// TIA Portal project "scl_5" (V18)

(* hardware
DEVICE "S7-1200 station_1"  S7-1200 Station
   slot 0: "Rack_0"  S7-1200 Rack  Rack  V1.0
   slot 1: "PLC_1"  CPU 1214C DC/DC/DC  6ES7 214-1AG40-0XB0  V4.6
*)

// ===== PLC "PLC_1"  CPU 1214C DC/DC/DC =====

VAR_GLOBAL   // PLC tag table "Default tag table"
   "İLERİ START" AT %I0.0 : Bool;
   "GERİ START" AT %I0.1 : Bool;
   "STOP" AT %I0.2 : Bool;
   "MOTOR İLERİ" AT %Q0.0 : Bool;
   "MOTOR GERİ" AT %Q0.1 : Bool;
END_VAR

FUNCTION "Block_1" : Void   // FC1, SCL
{ S7_Optimized_Access := 'TRUE' }
VERSION : 0.1
BEGIN
   IF "İLERİ START" AND NOT "MOTOR GERİ"=1 THEN
       // Statement section IF

       "MOTOR İLERİ":=1;
   END_IF;
   IF "GERİ START" AND NOT "MOTOR İLERİ" = 1 THEN
       // Statement section IF

       "MOTOR GERİ" := 1;

   END_IF;
   IF "STOP"=1 THEN
       // Statement section IF

       "MOTOR İLERİ" := 0;
       "MOTOR GERİ" := 0;
   END_IF;
END_FUNCTION

ORGANIZATION_BLOCK "Main"   // OB1, LAD, ProgramCycle
TITLE = "Main Program Sweep (Cycle)"
{ S7_Optimized_Access := 'TRUE' }
VERSION : 0.1
   VAR_INPUT
      Initial_Call : Bool;   // Initial call of this OB
      Remanence : Bool;   // =True, if remanent data are available
   END_VAR
BEGIN

REGION Network 1
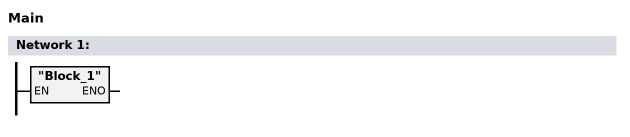
   RUNG wire#powerrail
      "Block_1"()
   END_RUNG
   // the same network as SCL:
   "Block_1"();
END_REGION
END_ORGANIZATION_BLOCK